FUNCTION_BLOCK FB_PMLStateLogger
VAR_IN_OUT
    a_fbPMLAlarms : ARRAY[1..48] OF FB_TcAlarm; //Array of alarms for Core PackML events that exist in any PackML enabled module
END_VAR
VAR_INPUT
    sModulePrefix  : STRING;       //Prefix String for all state change events (Typically the ID and Name of the module in some concatenated form)
    eState         : E_PMLState;   //Current PML state of the module
    bLogAllChanges : BOOL := TRUE; //If TRUE, all state change events will be logged, regardless of severity, otherwise info alarms are ignored
END_VAR
VAR_OUTPUT
END_VAR
VAR
    eLastState   : E_PMLState := E_PMLState.ePMLState_Aborted; //Saves the previous state each time the block is run
    refTempAlarm : REFERENCE TO FB_TcAlarm;                    //Temporary reference that makes severity checking simpler vs individually checking each change alarm within the case statement
END_VAR

IF eState <> eLastState THEN //If state has changed
    CASE eState OF           //Get the stored alarm that corresponds to the newly entered state and save its reference temporarily
        E_PMLState.ePMLState_Starting:
            refTempAlarm REF= a_fbPMLAlarms[E_PMLAlarms.StateStartingEnter];
        E_PMLState.ePMLState_Execute:
            refTempAlarm REF= a_fbPMLAlarms[E_PMLAlarms.StateExecuteEnter];
        E_PMLState.ePMLState_Completing:
            refTempAlarm REF= a_fbPMLAlarms[E_PMLAlarms.StateCompletingEnter];
        E_PMLState.ePMLState_Complete:
            refTempAlarm REF= a_fbPMLAlarms[E_PMLAlarms.StateCompleteEnter];
        E_PMLState.ePMLState_Resetting:
            refTempAlarm REF= a_fbPMLAlarms[E_PMLAlarms.StateResettingEnter];
        E_PMLState.ePMLState_Idle:
            refTempAlarm REF= a_fbPMLAlarms[E_PMLAlarms.StateIdleEnter];
        E_PMLState.ePMLState_Holding:
            refTempAlarm REF= a_fbPMLAlarms[E_PMLAlarms.StateHoldingEnter];
        E_PMLState.ePMLState_Held:
            refTempAlarm REF= a_fbPMLAlarms[E_PMLAlarms.StateHeldEnter];
        E_PMLState.ePMLState_Unholding:
            refTempAlarm REF= a_fbPMLAlarms[E_PMLAlarms.StateUnholdingEnter];
        E_PMLState.ePMLState_Suspending:
            refTempAlarm REF= a_fbPMLAlarms[E_PMLAlarms.StateSuspendingEnter];
        E_PMLState.ePMLState_Suspended:
            refTempAlarm REF= a_fbPMLAlarms[E_PMLAlarms.StateSuspendedEnter];
        E_PMLState.ePMLState_Unsuspending:
            refTempAlarm REF= a_fbPMLAlarms[E_PMLAlarms.StateUnsuspendingEnter];
        E_PMLState.ePMLState_Stopping:
            refTempAlarm REF= a_fbPMLAlarms[E_PMLAlarms.StateStoppingEnter];
        E_PMLState.ePMLState_Stopped:
            refTempAlarm REF= a_fbPMLAlarms[E_PMLAlarms.StateStoppedEnter];
        E_PMLState.ePMLState_Aborting:
            refTempAlarm REF= a_fbPMLAlarms[E_PMLAlarms.StateAbortingEnter];
        E_PMLState.ePMLState_Aborted:
            refTempAlarm REF= a_fbPMLAlarms[E_PMLAlarms.StateAbortedEnter];
        E_PMLState.ePMLState_Clearing:
            refTempAlarm REF= a_fbPMLAlarms[E_PMLAlarms.StateClearingEnter];
        E_PMLState.ePMLState_Undefined:
            refTempAlarm REF= a_fbPMLAlarms[E_PMLAlarms.StateUndefinedEnter];
    END_CASE

    //If the FB is set to log all changes, log the change, otherwise check the severity of the alarm and log it if it exceeds 'info' severity
    IF bLogAllChanges OR (refTempAlarm.eSeverity <> TcEventSeverity.Info AND refTempAlarm.eSeverity <> TcEventSeverity.Verbose) THEN
        refTempAlarm.Raise(0);
    END_IF

    CASE eLastState OF //Clear the previous state's event (Events will remain 'Raised' as long as the module remains in that state)
        E_PMLState.ePMLState_Starting:
            a_fbPMLAlarms[E_PMLAlarms.StateStartingEnter].Clear(0, 0);
        E_PMLState.ePMLState_Execute:
            a_fbPMLAlarms[E_PMLAlarms.StateExecuteEnter].Clear(0, 0);
        E_PMLState.ePMLState_Completing:
            a_fbPMLAlarms[E_PMLAlarms.StateCompletingEnter].Clear(0, 0);
        E_PMLState.ePMLState_Complete:
            a_fbPMLAlarms[E_PMLAlarms.StateCompleteEnter].Clear(0, 0);
        E_PMLState.ePMLState_Resetting:
            a_fbPMLAlarms[E_PMLAlarms.StateResettingEnter].Clear(0, 0);
        E_PMLState.ePMLState_Idle:
            a_fbPMLAlarms[E_PMLAlarms.StateIdleEnter].Clear(0, 0);
        E_PMLState.ePMLState_Holding:
            a_fbPMLAlarms[E_PMLAlarms.StateHoldingEnter].Clear(0, 0);
        E_PMLState.ePMLState_Held:
            a_fbPMLAlarms[E_PMLAlarms.StateHeldEnter].Clear(0, 0);
        E_PMLState.ePMLState_Unholding:
            a_fbPMLAlarms[E_PMLAlarms.StateUnholdingEnter].Clear(0, 0);
        E_PMLState.ePMLState_Suspending:
            a_fbPMLAlarms[E_PMLAlarms.StateSuspendingEnter].Clear(0, 0);
        E_PMLState.ePMLState_Suspended:
            a_fbPMLAlarms[E_PMLAlarms.StateSuspendedEnter].Clear(0, 0);
        E_PMLState.ePMLState_Unsuspending:
            a_fbPMLAlarms[E_PMLAlarms.StateUnsuspendingEnter].Clear(0, 0);
        E_PMLState.ePMLState_Stopping:
            a_fbPMLAlarms[E_PMLAlarms.StateStoppingEnter].Clear(0, 0);
        E_PMLState.ePMLState_Stopped:
            a_fbPMLAlarms[E_PMLAlarms.StateStoppedEnter].Clear(0, 0);
        E_PMLState.ePMLState_Aborting:
            a_fbPMLAlarms[E_PMLAlarms.StateAbortingEnter].Clear(0, 0);
        E_PMLState.ePMLState_Aborted:
            a_fbPMLAlarms[E_PMLAlarms.StateAbortedEnter].Clear(0, 0);
        E_PMLState.ePMLState_Clearing:
            a_fbPMLAlarms[E_PMLAlarms.StateClearingEnter].Clear(0, 0);
        E_PMLState.ePMLState_Undefined:
            a_fbPMLAlarms[E_PMLAlarms.StateUndefinedEnter].Clear(0, 0);

    END_CASE

    eLastState := eState; //Store previous state
END_IF

END_FUNCTION_BLOCK

(* stored: Version 1.1.0.1, ProductVersion 3.1.4024.11
   POU FB_PMLStateLogger: Id {8b359582-8387-45ce-89d5-2a1b5888ef7a}, SpecialFunc None *)
